PROGRAM MAIN
VAR
	// Data Recording
	fbUR5tcp : FB_RobotTCPReceive := (Robot := 'UR5');
	fbUR3tcp : FB_RobotTCPReceive := (Robot := 'UR3');
	eRobotDataRecordingState : E_RobotDataRecordingStates;
	
	
	// Optoforce
	fbRecFTData : FB_FT_UDPConnection;

	
	// Triggers
	StartTrig: R_TRIG;
	StopTrig: F_TRIG;
	
	// Procees State Machine
	eProcessMode : E_ProcessModes;
	sProcessState : STRING;
	

	
END_VAR

(* =======================================================
Update veriables on every cycle
======================================================= *)
// Record time every cycle
Global.nCurrentTime := F_GetSystemTime();

// Triggers for start and stop buttons on control pendant
StartTrig(CLK := Global.pbStart); // Start
StopTrig(CLK := Global.pbStop); // Stop

(* =======================================================
Process Mode State Machine 
======================================================= *)
// Interrupts
	// Stop Button
	IF StopTrig.Q OR Global.bCycleStop THEN 
		eProcessMode := E_ProcessModes.Stopping;
		Global.bCycleStop := FALSE;
	END_IF
// State Machine
CASE eProcessMode OF
	E_ProcessModes.Idle:
		sProcessState := 'Idle';
		// Wait for start button to trigger
		IF StartTrig.Q OR Global.bCycleStart THEN
			eProcessMode := E_ProcessModes.Running;
			Global.bCycleStart := FALSE;
		END_IF
		Global.indStartPB := FALSE;
		Global.indStopPB := TRUE;
		
	E_ProcessModes.Running:
		sProcessState := 'Assigning Tasks';
		Global.bActivateTaskAssignment := TRUE;
		Global.indStartPB := TRUE;
		Global.indStopPB := FALSE;
	E_ProcessModes.Stopping:
		sProcessState := 'Performing Last Tasks';
		Global.bActivateTaskAssignment := FALSE;
		eProcessMode := E_ProcessModes.Idle;
END_CASE

(* =======================================================
Data Collection Processes
======================================================= *)


// Enable TCP/IP Data collection from robots
fbUR5tcp.bEnable := Global.bActivateTCPIPDataCollection;
fbUR3tcp.bEnable := Global.bActivateTCPIPDataCollection;
IF Global.bActivateTCPIPDataCollection THEN
	fbUR5tcp.bRecordData := Global.bActivateTCPIPDataRecording;
	fbUR3tcp.bRecordData := Global.bActivateTCPIPDataRecording;
ELSE
	fbUR5tcp.bRecordData := FALSE;
	fbUR3tcp.bRecordData := FALSE;
END_IF


// Enable UDP Data collection from Force and Torque Sensor
fbRecFTData.bEnable := Global.bActivateFTDataCollection;
IF Global.bActivateFTDataCollection THEN
	fbRecFTData.bRecordData := Global.bActivateFTDataRecording;
ELSE
	fbRecFTData.bRecordData := FALSE;
END_IF

(* =======================================================
Function block Calls
======================================================= *)
fbUR5tcp();
fbUR3tcp();
fbRecFTData(stOptoforceData => Global.stFTData );

(* =======================================================
Sub-programs that run all the time
======================================================= *)
P_Safety(); // Handle Safety Funftions and collects safety related data
P_InputOutputHandling();
P_TaskHandling();

(* =======================================================
Automated Experiment Data Cleaning / Reset
======================================================= *)
IF Global.bResetPartCount THEN
	Global.nPartsStarted := 0;
	Global.nPartsCompleted := 0;
	Global.nTotalPartTime := 0;
	Global.nAveragePartTime := 0;
	Global.bResetPartCount := FALSE;
END_IF

END_PROGRAM

(* stored: Version 1.1.0.1, ProductVersion 3.1.4020.12
   POU MAIN: Id {5c12abd9-0d27-431f-9a5a-1bee0375886f}, SpecialFunc None *)
